{attribute addProperty BoxType "EK1100-0000-0018"}
{attribute addProperty Id "Beckhoff_ELM37xxEK1122Beckhoff_ELM37xxEK1122_FB33499C162A_0001_ELM3702_0000_0016ELM3702_08F8D9E433842.25A_0002_ELM3702_0000_0017ELM3702_08F8D9E433842.25A_0003_ELM3704_0000_0016ELM3704_B740F21646658.25A_0004_ELM3704_0000_0017ELM3704_B740F21646658.25A_0005_ELM3704_0001_0017ELM3704_B740F21646658.25A_0006_ELM3704_0020_0016ELM3704_B740F21646658.25A_0007_ELM3702_0101_0016ELM3702_08F8D9E433842.25A_0008_ELM3704_1001_0016ELM3704_B740F21646658.25A_0009_ELM3704_1001_0017ELM3704_B740F21646658.25"}
{attribute addProperty CRC "937131418"}
{attribute addProperty SizeInBites "3826"}
{attribute addProperty SizeInBytes "478.25"}
TYPE Beckhoff_ELM37xx_37DB7D9A EXTENDS EK1100_179A0949 :
STRUCT
	{attribute addProperty Name "Beckhoff_ELM37xxEK1122"}
	Beckhoff_ELM37xxEK1122 : Beckhoff_ELM37xxEK1122_FB33499C;
	{attribute addProperty Name "A_0001_ELM3702_0000_0016"}
	A_0001_ELM3702_0000_0016 : ELM3702_08F8D9E4;
	{attribute addProperty Name "A_0002_ELM3702_0000_0017"}
	A_0002_ELM3702_0000_0017 : ELM3702_08F8D9E4;
	{attribute addProperty Name "A_0003_ELM3704_0000_0016"}
	A_0003_ELM3704_0000_0016 : ELM3704_B740F216;
	{attribute addProperty Name "A_0004_ELM3704_0000_0017"}
	A_0004_ELM3704_0000_0017 : ELM3704_B740F216;
	{attribute addProperty Name "A_0005_ELM3704_0001_0017"}
	A_0005_ELM3704_0001_0017 : ELM3704_B740F216;
	{attribute addProperty Name "A_0006_ELM3704_0020_0016"}
	A_0006_ELM3704_0020_0016 : ELM3704_B740F216;
	{attribute addProperty Name "A_0007_ELM3702_0101_0016"}
	A_0007_ELM3702_0101_0016 : ELM3702_08F8D9E4;
	{attribute addProperty Name "A_0008_ELM3704_1001_0016"}
	A_0008_ELM3704_1001_0016 : ELM3704_B740F216;
	{attribute addProperty Name "A_0009_ELM3704_1001_0017"}
	A_0009_ELM3704_1001_0017 : ELM3704_B740F216;
END_STRUCT
END_TYPE

(* stored: Version 1.2.0.0, ProductVersion 3.1.4024.9
   DUT Beckhoff_ELM37xx_37DB7D9A: Id {f867e5ad-2767-41ef-94f3-e5412cb25d0f} *)
